FUNCTION_BLOCK NormallyOpenPushButton IMPLEMENTS I_PushButton

VAR
	Input	AT %I* : BOOL; 
END_VAR

PROPERTY IsPressed : BOOL
GET
IsPressed := Input;
END_GET
END_PROPERTY

PROPERTY IsReleased : BOOL
GET
IsReleased := NOT IsPressed;
END_GET
END_PROPERTY

END_FUNCTION_BLOCK

(* stored: Version 1.1.0.1, ProductVersion 3.1.4024.12
   POU NormallyOpenPushButton: Id {23008e7e-5bcc-42a3-9965-5e73ef7363ea}, SpecialFunc None
   Property IsPressed: Id {2f220a47-b3de-4ebd-bcc7-8b3116a8033d}
   Get Get: Id {157cf45b-07de-492f-84cf-2f953c550b82}
   Property IsReleased: Id {ef17f393-5d62-40b9-b096-df58a44a0395}
   Get Get: Id {5ac33980-0d1c-493b-ad46-0fb863c9929b} *)
